// TIA Portal V19 export
TYPE "LAF_typeXXXXParameters"
// stored: Access Published
   STRUCT
      manual : "LAF_typeXXXMannualParameters";
      production : "LAF_typeXXXProductionParameters";
      maintenance { S7_SetPoint := 'True'} : "LAF_typeXXXMaintanceParameters";
   END_STRUCT;
END_TYPE
